// TIA Portal V19 export
TYPE "LEXCHANGETRAY_typeNgConveyor_signalTM_Cmd"
// stored: Access Published
   STRUCT
      simActive : Bool;
   END_STRUCT;
END_TYPE
